// TwinCAT 3 PLC project OpenbareToilet
// ProgramVersion: 3.1.4024.0
// libraries:
//   Tc2_Standard, * (Beckhoff Automation GmbH)
//   Tc2_System, * (Beckhoff Automation GmbH)
//   Tc3_Module, * (Beckhoff Automation GmbH)
// project tree:
//   / PlcTask.TcTTO
//   POUs/ MAIN.TcPOU
// (motion and I/O tree: see PLC project trappenhuis_extraverlenging)
// real-time tasks:
//   TASK PlcTask: cycle T#10ms, priority 20, ADS port 350
//   TASK PlcTask1: cycle T#10ms, priority 21, ADS port 351
//   TASK PlcTask2: cycle T#10ms, priority 22, ADS port 352
//   TASK PlcTask3: cycle T#10ms, priority 23, ADS port 353
//   TASK PlcTask4: cycle T#10ms, priority 24, ADS port 354
//   TASK PlcTask5: cycle T#10ms, priority 25, ADS port 355
//   TASK PlcTask6: cycle T#10ms, priority 26, ADS port 356
//   TASK PlcTask7: cycle T#10ms, priority 27, ADS port 357
//   TASK PlcTask8: cycle T#10ms, priority 28, ADS port 358
//   TASK PlcTask9: cycle T#10ms, priority 29, ADS port 359
//   TASK PlcTask10: cycle T#10ms, priority 30, ADS port 360

CONFIGURATION OpenbareToilet
    RESOURCE PLC ON TwinCAT3
        TASK PlcTask(INTERVAL := T#10ms, PRIORITY := 24);
        PROGRAM MAIN WITH PlcTask : MAIN;
    END_RESOURCE
END_CONFIGURATION

// ---- POUs/MAIN.TcPOU
PROGRAM MAIN
VAR
	S01, S02, S03: BOOL; // Bistabiele schakelaars voor de toiletten
	L01, L02, L03: BOOL; // Lampen voor de toiletten
	Ventilator: BOOL; // Gemeenschappelijke ventilator
	fbVentilatorTimer: TOF; // Timer voor de ventilator
END_VAR

(*
Openbaar toilet (4 regel code)

Er zijn drie toiletten met elk een lamp voor de verlichting (L01, L02 en L03) en elk een bistabiele schakelaar
(S01, S02 en S03) om deze lampen respectievelijk aan te steken.
 Wanneer iemand een toilet binnengaat en de schakelaar bedient gebeuren twee zaken:

    enkel in het betreffende toilet zal de lamp gaan branden
    er is ook één gemeenschappelijke ventilator voor het verluchten van de
    toiletten, deze ventilator zal in werking treden als eender welke
    schakelaar wordt bediend.

Als de bezoeker terug buitengaat en de verlichting uitschakelt gebeuren twee zaken:

    in het betreffende toilet zal de lamp uitgeschakeld worden
    de gemeenschappelijke ventilator zal nog 2 minuten (simuleer 5
    seconden) blijven werken en daarna automatisch uitschakelen (op
    voorwaarde dat intussen niemand anders de toiletten bezoekt).
*)

L01 := S01; L02 := S02; L03 := S03; // Bediening lampen
Ventilator := S01 OR S02 OR S03 OR fbVentilatorTimer.Q; // Ventilator werkt als een van de schakelaars is ingeschakeld of de timer loopt
fbVentilatorTimer(IN:=S01 OR S02 OR S03, PT:=T#5s); // Timer start als een van de schakelaars wordt ingeschakeld, looptijd 5 seconden

END_PROGRAM
